FUNCTION_BLOCK FB_PowerModule
VAR_IN_OUT CONSTANT
	st_params							: ST_PowerModule_params;
	st_calibration						: ST_PowerModule_Calibration;
END_VAR


VAR_INPUT
	set									: ST_PowerModule_set; //only setteable from intern powerstack function
	r_batteryDCVoltage					: REAL;
	b_enable							: BOOL;
	e_ID								: eObject_ID;
END_VAR

VAR_OUTPUT
	{attribute 'TcAnalytics'}
	get									: ST_PowerModule_get;
	b_MccbEDM							: BOOL;
END_VAR	

VAR									
	Inverter							: FB_PowerModule_Inverter();
	Buscoupler							: FB_PowerModule_Buscoupler();
	ton_ResetPulse						: TON := (PT:= T#100MS);
	
	r_Prq: REAL;
	r_Qrq: REAL;
	pin: REAL;
	QIN: REAL;
END_VAR

IF b_enable THEN
	get.b_online := get.ui_buscouplerCommStatus = 0 AND get.ui_InverterCommStatus = 0;
	
	//Instantiate function blocks
	Buscoupler(get:=get, b_MccbEDM := b_MccbEDM, b_D7SyncRq := set.b_D7SyncRequest);
	Inverter(set := set, get:=get, st_params:=st_params);
	//defaults
	Inverter.ControlWord.b_FieldbusControlEnable := st_params.b_FieldBusControlEnable;

	//Control fan contactor.
	FanControl(st_params := st_params);
	
	//Set PowerModule status
	GetPowerModuleStatus();
	
	//Set DroopLimit
	SetInverterSettings();
	
	//Calculate derivatives
	CalculateDerivativePowerValues();
	
	//Parallel Drive
	SetParallelDrive();
	
	//setEvents
	SetEvents(events := get.Events, st_params:=st_Params);
	
	//FILL GET STRUCT
	GetInverterModes();
	FillAdditionalGets(get, set);
	
	//inverter.ControlWord.b_Reset := FALSE;
	
	SetParallelDrive();
	
	IF get.StatusWord.b_Fault THEN
		Shutdown(TRUE);
	END_IF
	
	IF GVL.b_initCycle THEN
		init();
	END_IF
END_IF

r_Prq := CompensationCurve(PIN := pin, QIN := qin, coef := st_calibration.PCoefficients, mode := 0);
r_Qrq := CompensationCurve(PIN := pin, QIN := qin, coef := st_calibration.QCoefficients, mode := 1);

METHOD BaseValueToRef : REAL;
VAR_INPUT
	IN : REAL;
END_VAR
BaseValueToRef:= IN / MAX(1, st_params.r_InverterRatedCurrent) * 100;
END_METHOD

METHOD PRIVATE CalculateDerivativePowerValues : BOOL
get.r_ReactivePower	:= get.r_ACVoltageD7 * 1.73 * get.r_ReactiveCurrent / 1000; // kvar
get.r_ActivePower	:= get.r_ACVoltageSupply* 1.73 * get.r_activeCurrent / 1000;
get.r_ApparentPower	:= SQRT(MAX(0,EXPT(get.r_ActivePower,2) + EXPT(get.r_ReactivePower,2)));
get.r_LoadPercent	:= get.r_ACCurrent / MAX(1, st_params.r_InverterRatedCurrent) * 100;
get.r_DCPower		:= get.r_DCCurrent * get.r_DCVoltage / 1000; // kW
END_METHOD

METHOD CheckDCVoltage : BOOL

VAR_INST
	b_DCprechargeOK				: BOOL; 
	b_DCVoltageOK				: BOOL;
	ton_DCOKreleaseTime			: TON := (PT:= T#1S);
END_VAR
b_DCPrechargeOK := ABS(r_BatteryDCVoltage - get.r_DCVoltage) <=  st_params.ui_DCVoltageDeltaPrechargeOK;
b_DCVoltageOK := get.r_DCVoltage > st_params.ui_DCvoltageMinPrechargeOK;

ton_DCOKReleaseTime(IN:= b_DCPrechargeOK AND b_DCVoltageOK);

CheckDCVoltage :=ton_DCOKReleaseTime.Q;
END_METHOD

METHOD CompensationCurve : REAL
VAR_INPUT
	PIN			: REAL; 
	QIN			: REAL;
	mode		: BYTE; // 0 = Pout, 1 = Qout;
END_VAR

VAR_IN_OUT CONSTANT
	coef : ST_Powermodule_PowerCurveCoefficients;
END_VAR

VAR_INST
	Q1			: REAL;
	Q2			: REAL;
	disc 		: REAL;
	Avalues		: REAL;
	Bvalues		: REAL;
	Cvalues		: REAL;
	depVar		: REAL;
	indepVar	: REAL;
END_VAR
IF NOT coef.enable THEN
	CompensationCurve := SEL(mode =0, Qin, Pin);
	RETURN; // Geen reële oplossing
END_IF


IF mode = 0 THEN
	indepVar := Pin;
	depVar := Qin;

ELSE
	indepVar := Qin;
	depVar := Pin;
END_IF

Avalues := coef.a;
BValues := coef.c*depVar + coef.d;
CValues := coef.b*EXPT(depVar,2)+coef.e*depVar + coef.f - indepVar;

disc := EXPT(BValues,2)-(4*AValues*CValues);
IF disc < 0 THEN
	CompensationCurve := indepVar;
	RETURN; // Geen reële oplossing
END_IF

// Controleer discriminant
IF Avalues = 0 THEN
    // Lineaire oplossing: B * P + C = 0 → P = -C / B
    IF BValues = 0 THEN
        RETURN; // onoplosbaar
    ELSE
        CompensationCurve := -CValues / BValues;
        RETURN;
    END_IF
END_IF

// Kwadratische oplossing (ABC)
Q1 := (-BValues + SQRT(disc)) / (2 * Avalues);
Q2 := (-BValues - SQRT(disc)) / (2 * Avalues);
CompensationCurve := Q1;
//// Kies de beste wortel (voorbeeld: dichtsbijzijnde bij indepVar)
//IF ABS(Q1 - indepVar) < ABS(Q2 - indepVar) THEN
//    CompensationCurve := Q1;
//ELSE
//    CompensationCurve := Q2;
//END_IF
END_METHOD

METHOD PRIVATE CoupleDC : BOOL
VAR_INPUT
END_VAR
IF get.StatusWord.b_ReadyToDCCharge THEN
	buscoupler.b_DCprechargeContactor := TRUE;
	buscoupler.b_DCMainContactor := CheckDCvoltage();
	CoupleDC := get.b_DCcontactorFb;
END_IF
END_METHOD

METHOD PRIVATE DecoupleDC : BOOL

VAR_INST
	b_DCmainreleaseConditionOK 	:  BOOL;
	b_DCprereleaseConditionOK 	:  BOOL;
	ton_PrechargeReleaseDelay	:  TON := (PT:= T#1S);
END_VAR

VAR
	r_DCreleaseCurrent		: REAL := 5;
	r_DCreleaseVoltage		: REAL := 10;
END_VAR
// Release main contactor first based on current
b_DCmainreleaseConditionOK := ABS(get.r_DCCurrent) < r_DCreleaseCurrent AND NOT get.StatusWord.b_Running;
IF b_DCmainreleaseConditionOK THEN
	buscoupler.b_DCmainContactor := FALSE;
END_IF

// release precharge based on voltage contactor 
b_DCprereleaseConditionOK := NOT get.b_DCcontactorFb OR r_batteryDCVoltage < r_DCreleaseVoltage; //NOT get.b_DCcontactorFb (Not for units without precharge, rewire output4 to input 4 of buscoupler.)
ton_PrechargeReleaseDelay(IN:= b_DCprereleaseConditionOK); //some delay added to be sure
IF ton_PrechargeReleaseDelay.Q THEN
	buscoupler.b_DCprechargeContactor := FALSE;
END_IF 

//Give feedback
IF b_DCprereleaseConditionOK AND b_DCmainreleaseConditionOK THEN
	DecoupleDc := NOT buscoupler.b_DCprechargeContactor AND NOT get.b_DCcontactorFb;
END_IF
END_METHOD

METHOD PRIVATE FanControl : BOOL
VAR_IN_OUT CONSTANT
	st_params : ST_Powermodule_params;
END_VAR
	


VAR_INST
	b_fanOn				: BOOL;
	tof_FanOffDelay		: TOF := (PT := T#60S);
END_VAR
IF get.r_TemperatureMax > st_params.r_TempFanOn OR get.r_LoadPercent > st_params.r_powerLoadFanOn THEN
	b_fanOn := TRUE;
ELSIF get.r_TemperatureMax < st_params.r_TempFanOn - 5 AND get.r_LoadPercent < st_params.r_powerLoadFanOn - 10 THEN
	b_fanOn := FALSE;
END_IF


tof_FanOffDelay(
	IN:= b_fanOn);
	
buscoupler.b_FanOn := set.b_FanContactor OR tof_FanOffDelay.Q;
END_METHOD

METHOD FillAdditionalGets : BOOL
VAR_IN_OUT
		get : ST_Powermodule_get;
		set	: ST_Powermodule_set;
END_VAR
get.r_TemperatureMax := GetMaxTemperature();
get.r_Pset := set.r_ActivePower;
get.r_Qset := set.r_ReactivePower;
get.b_PrechargeContactor := buscoupler.b_DCprechargeContactor;
END_METHOD

METHOD GetDiagnostics 
VAR_IN_OUT
	AddError		: ARRAY [*] OF FB_AddErrorST;
	a_ActiveEvents	: ARRAY [*] OF ST_ErrorStruct;
	w_Index			: WORD;
END_VAR

VAR
	by_errCt	: BYTE;
	by_warnCt	: BYTE;
END_VAR


VAR_INST
	b_test: BOOL;
END_VAR
(*POWERMODULE*)
	//Inverter faults
	(*OverCurr Fault*)		AddError[w_Index](
			b_ErrorTrig			:= Get.Events.b_F1OverCurrent,
			out_ST_Error			:= a_ActiveEvents[w_Index],
			w_ErrorID					:= 1,
			e_objectID				:= e_ID,
			s_Message				:= 'overcurrent fault (F1)',
			e_sev					:= eSeverity.Quickshutdown,
			);
		IF AddError[w_Index].b_out THEN by_errCt := by_errCt + 1; END_IF;
		w_Index := w_Index +1;
		
	(*OverVolt Fault*)		AddError[w_Index](
			b_ErrorTrig			:= Get.Events.b_F2OverVoltage,
			out_ST_Error			:= a_ActiveEvents[w_Index],
			w_ErrorID					:= 2,
			s_Message				:= 'DC overvoltage fault (F2)',
			e_sev					:= eSeverity.Quickshutdown,
			);
		IF AddError[w_Index].b_out THEN by_errCt := by_errCt + 1; END_IF;
		w_Index := w_Index +1;
	
	(*UnderVolt Fault*)		AddError[w_Index](
			b_ErrorTrig			:= Get.Events.b_F9UnderVoltage,
			out_ST_Error			:= a_ActiveEvents[w_Index],
			w_ErrorID					:= 3,
			s_Message				:= 'DC undervoltage fault (F9)',
			e_sev					:= eSeverity.Quickshutdown,
			);
		IF AddError[w_Index].b_out THEN by_errCt := by_errCt + 1; END_IF;
		w_Index := w_Index +1;
	
	(*ShortCurr Fault*)		AddError[w_Index](
			b_ErrorTrig		:= Get.Events.b_F91ShortCircuit,
			out_ST_Error			:= a_ActiveEvents[w_Index],
			w_ErrorID					:= 4,
			s_Message				:= 'short circuit fault (F91)',
			e_sev					:= eSeverity.Quickshutdown,
			);
		IF AddError[w_Index].b_out THEN by_errCt := by_errCt + 1; END_IF;
		w_Index := w_Index +1;
		
	(*Earth Fault*)			AddError[w_Index](
			b_ErrorTrig		:= Get.Events.b_F3EarthFault,
			out_ST_Error			:= a_ActiveEvents[w_Index],
			w_ErrorID					:= 5,
			s_Message				:= 'earth fault (F3)',
			e_sev					:= eSeverity.Quickshutdown,
			);
		IF AddError[w_Index].b_out THEN by_errCt := by_errCt + 1; END_IF;
		w_Index := w_Index +1;
		
	(*LineSync Fault*)		AddError[w_Index](
			b_ErrorTrig		:= Get.Events.b_F10LineSynchFault,
			out_ST_Error			:= a_ActiveEvents[w_Index],
			w_ErrorID					:= 6,
			s_Message				:= 'line synchronisation fault (F10)',
			e_sev					:= eSeverity.Quickshutdown,
			);
		IF AddError[w_Index].b_out THEN by_errCt := by_errCt + 1; END_IF;
		w_Index := w_Index +1;
	
	(*Keypad Fault*)		AddError[w_Index](
			b_ErrorTrig		:= Get.Events.b_F52KeypadOCCommFault,
			out_ST_Error			:= a_ActiveEvents[w_Index],
			w_ErrorID					:= 7,
			s_Message				:= 'keypad communication fault (F52)',
			e_sev					:= eSeverity.warning,
			);
		IF AddError[w_Index].b_out THEN by_errCt := by_errCt + 1; END_IF;
		w_Index := w_Index +1;
	
	(*Fieldbus Fault*)		AddError[w_Index](
			b_ErrorTrig		:= Get.Events.b_F53FieldbusFault,
			out_ST_Error			:= a_ActiveEvents[w_Index],
			w_ErrorID					:= 8,
			s_Message				:= 'fieldbus fault (F53)',
			e_sev					:= eSeverity.Quickshutdown,
			);
		IF AddError[w_Index].b_out THEN by_errCt := by_errCt + 1; END_IF;
		w_Index := w_Index +1;
		
	(*Systembus Fault*)		AddError[w_Index](
			b_ErrorTrig		:= Get.Events.b_F59SystembusFault,
			out_ST_Error			:= a_ActiveEvents[w_Index],
			w_ErrorID					:= 9,
			s_Message				:= 'system bus Fault (F59)',
			e_sev					:= eSeverity.Quickshutdown,
			);
		IF AddError[w_Index].b_out THEN by_errCt := by_errCt + 1; END_IF;
		w_Index := w_Index +1;
	
	(*IOslot Fault*)		AddError[w_Index](
			b_ErrorTrig		:= Get.Events.b_F54SlotCommunicationFault,
			out_ST_Error			:= a_ActiveEvents[w_Index],
			w_ErrorID					:= 10,
			s_Message				:= 'IO slot communication fault (F54)',
			e_sev					:= eSeverity.Quickshutdown,
			);
		IF AddError[w_Index].b_out THEN by_errCt := by_errCt + 1; END_IF;
		w_Index := w_Index +1;
		
	(*4ma meas Fault*)		AddError[w_Index](
			b_ErrorTrig		:= Get.Events.b_F50Meas4mAFault,
			out_ST_Error			:= a_ActiveEvents[w_Index],
			w_ErrorID					:= 11,
			s_Message				:= 'measurement 4 mA fault (F50)',
			e_sev					:= eSeverity.info,
			b_AutoClear			:= TRUE,
		);
		w_Index := w_Index +1;
		
	(*Watchdog Fault*)		AddError[w_Index](
			b_ErrorTrig		:= Get.Events.b_WatchdogError,
			out_ST_Error			:= a_ActiveEvents[w_Index],
			w_ErrorID					:= 12,
			s_Message				:= 'watchdog fault',
			e_sev					:= eSeverity.Quickshutdown,
			);
		IF AddError[w_Index].b_out THEN by_errCt := by_errCt + 1; END_IF;
		w_Index := w_Index +1;
	
	(*Mccb Trip*)			AddError[w_Index](
			b_ErrorTrig			:= FALSE, //Get.Events.b_MCCBtrip,
			out_ST_Error			:= a_ActiveEvents[w_Index],
			w_ErrorID					:= 13,
			s_Message				:= 'MCCB trip',
			e_sev					:= eSeverity.warning
		);
		w_Index := w_Index +1;

	(*Shutdown TimeOut*)			AddError[w_Index](
			b_ErrorTrig			:= Get.Events.b_ShutdownTimeOut,
			out_ST_Error			:= a_ActiveEvents[w_Index],
			w_ErrorID					:= 14,
			s_Message				:= 'shutdown Timeout',
			e_sev					:= eSeverity.QuickShutdown
		);
		w_Index := w_Index +1;
		
	(*output phase fault (F11)*)	AddError[w_Index](
			b_ErrorTrig				:= Get.Events.b_F11OutputPhaseFault,
			out_ST_Error			:= a_ActiveEvents[w_Index],
			w_ErrorID				:= 15,
			s_Message				:= 'output phase fault (F11)',
			e_sev					:= eSeverity.Quickshutdown
		);
		w_Index := w_Index +1;
		
	(*charge fault (F80)*)			AddError[w_Index](
			b_ErrorTrig				:= Get.Events.b_F80ChargeFault,
			out_ST_Error			:= a_ActiveEvents[w_Index],
			w_ErrorID				:= 16,
			s_Message				:= 'charge fault (F80)',
			e_sev					:= eSeverity.Quickshutdown
		);
		w_Index := w_Index +1;
		
		(*charge fault (F80)*)			AddError[w_Index](
			b_ErrorTrig				:= Get.Events.b_F51ExternalFault,
			out_ST_Error			:= a_ActiveEvents[w_Index],
			w_ErrorID				:= 17,
			s_Message				:= 'external fault (F51)',
			e_sev					:= eSeverity.Quickshutdown
		);
		w_Index := w_Index +1;
		
		(*IGBT fault (F31)*)		AddError[w_Index](
			b_ErrorTrig				:= Get.Events.b_F31IGBTFault,
			out_ST_Error			:= a_ActiveEvents[w_Index],
			w_ErrorID				:= 18,
			s_Message				:= 'IGBT fault (F31)',
			e_sev					:= eSeverity.Quickshutdown
		);
		w_Index := w_Index +1;
		
		(*MCB state fault (F64)*)		AddError[w_Index](
			b_ErrorTrig				:= Get.Events.b_F64MCBstateFault,
			out_ST_Error			:= a_ActiveEvents[w_Index],
			w_ErrorID				:= 19,
			s_Message				:= 'MCB state fault (F64)',
			e_sev					:= eSeverity.Quickshutdown
		);
		w_Index := w_Index +1;
	
	//Temperature Faults
	(*Gridch L1 Alarm*)		AddError[w_Index](
			b_ErrorTrig		:= Get.Events.b_CMChokeTemperatureTooHigh[1],
			out_ST_Error			:= a_ActiveEvents[w_Index],
			w_ErrorID					:= 20 ,
			s_Message				:= 'gridchoke L1 temperature too high',
			e_sev					:= eSeverity.normalshutdown,
			);
		IF AddError[w_Index].b_out THEN by_errCt := by_errCt + 1; END_IF;
		w_Index := w_Index +1;
		
	(*Gridch L2 Alarm*)		AddError[w_Index](
			b_ErrorTrig		:= Get.Events.b_CMChokeTemperatureTooHigh[2], //phase 2
			out_ST_Error			:= a_ActiveEvents[w_Index],
			w_ErrorID					:= 21 ,
			s_Message				:= 'gridchoke L2 temperature too high',
			e_sev					:= eSeverity.normalshutdown,
			);
		IF AddError[w_Index].b_out THEN by_errCt := by_errCt + 1; END_IF;
		w_Index := w_Index +1;
		
	(*Gridch L3 Alarm*)		AddError[w_Index](
			b_ErrorTrig		:= Get.Events.b_CMChokeTemperatureTooHigh[3], //phase 3
			out_ST_Error			:= a_ActiveEvents[w_Index],
			w_ErrorID					:= 22 ,
			s_Message				:= 'gridchoke L3 temperature too high',
			e_sev					:= eSeverity.normalshutdown,
			);
		IF AddError[w_Index].b_out THEN by_errCt := by_errCt + 1; END_IF;
		w_Index := w_Index +1;
		
	(*CMch L1 Alarm*)		AddError[w_Index](
			b_ErrorTrig		:= Get.Events.b_GridChokeTemperatureTooHigh[1], //phase 1
			out_ST_Error			:= a_ActiveEvents[w_Index],
			w_ErrorID					:= 23 ,
			s_Message				:= 'CM choke L1 temperature too high',
			e_sev					:= eSeverity.normalshutdown,
			);
		IF AddError[w_Index].b_out THEN by_errCt := by_errCt + 1; END_IF;
		w_Index := w_Index +1;
		
	(*CMch L2 Alarm*)		AddError[w_Index](
			b_ErrorTrig		:= Get.Events.b_CMChokeTemperatureTooHigh[2], //phase 2
			out_ST_Error			:= a_ActiveEvents[w_Index],
			w_ErrorID					:= 24 ,
			s_Message				:= 'CM choke L2 temperature too high',
			e_sev					:= eSeverity.normalshutdown,
			);
		IF AddError[w_Index].b_out THEN by_errCt := by_errCt + 1; END_IF;
		w_Index := w_Index +1;
		
	(*CMch L3 Alarm*)		AddError[w_Index](
			b_ErrorTrig		:= Get.Events.b_CMChokeTemperatureTooHigh[3], //phase 3
			out_ST_Error			:= a_ActiveEvents[w_Index],
			w_ErrorID					:= 25 ,
			s_Message				:= 'CM choke L3 temperature too high',
			e_sev					:= eSeverity.normalshutdown,
			);
		IF AddError[w_Index].b_out THEN by_errCt := by_errCt + 1; END_IF;
		w_Index := w_Index +1;
		
	(*CMch DC Alarm*)		AddError[w_Index](
			b_ErrorTrig		:= Get.Events.b_CMChokeTemperatureTooHigh[4], //DC
			out_ST_Error			:= a_ActiveEvents[w_Index],
			w_ErrorID					:= 26 ,
			s_Message				:= 'CM choke DC temperature too high',
			e_sev					:= eSeverity.normalshutdown,
			);
		IF AddError[w_Index].b_out THEN by_errCt := by_errCt + 1; END_IF;
		w_Index := w_Index +1;
		
	(*Inverter Alarm*)		AddError[w_Index](
			b_ErrorTrig		:= Get.Events.b_F14UnitOverTemperature,
			out_ST_Error			:= a_ActiveEvents[w_Index],
			w_ErrorID					:= 27 ,
			s_Message				:= 'overtemperature fault (F14)',
			e_sev					:= eSeverity.Quickshutdown
		);
		IF AddError[w_Index].b_out THEN by_errCt := by_errCt + 1; END_IF;
		w_Index := w_Index +1;	
		
	(*PT100 Fault*)			AddError[w_Index](
			b_ErrorTrig		:= Get.Events.b_F56TemperatureFault, //inverter Pt100 measurement
			out_ST_Error			:= a_ActiveEvents[w_Index],
			w_ErrorID					:= 28 ,
			s_Message				:= 'pt100 temperature fault (F56)',
			e_sev					:= eSeverity.normalshutdown,
			);
		IF AddError[w_Index].b_out THEN by_errCt := by_errCt + 1; END_IF;
		w_Index := w_Index +1;
		
	
	//Temperature Warnings
	(*Gridch L1 Warning*)	AddError[w_Index](
			b_ErrorTrig			:= Get.Events.b_gridChokeTemperatureHigh[1], //phase 1
			out_ST_Error			:= a_ActiveEvents[w_Index],
			w_ErrorID					:= 40 ,
			s_Message				:= 'gridchoke L1 temperature high',
			e_sev					:= eSeverity.warning,
			b_AutoClear			:= TRUE,
			);
		IF AddError[w_Index].b_out THEN by_warnCt := by_warnCt + 1; END_IF;
		w_Index := w_Index +1;
		
	(*Gridch L2 Warning*)	AddError[w_Index](
			b_ErrorTrig		:= Get.Events.b_GridchokeTemperatureHigh[2], //phase 2
			out_ST_Error			:= a_ActiveEvents[w_Index],
			w_ErrorID					:= 41 ,
			s_Message				:= 'gridchoke L2 temperature high',
			e_sev					:= eSeverity.warning,
			b_AutoClear			:= TRUE,
			);
		IF AddError[w_Index].b_out THEN by_warnCt := by_warnCt + 1; END_IF;
		w_Index := w_Index +1;
		
	(*Gridch L3 Warning*)	AddError[w_Index](
			b_ErrorTrig		:= Get.Events.b_GridChokeTemperatureHigh[3], //phase 3
			out_ST_Error			:= a_ActiveEvents[w_Index],
			w_ErrorID					:= 42 ,
			s_Message				:= 'gridchoke L3 temperature high',
			e_sev					:= eSeverity.warning,
			b_AutoClear			:= TRUE,
			);
		IF AddError[w_Index].b_out THEN by_warnCt := by_warnCt + 1; END_IF;
		w_Index := w_Index +1;
		
	(*CMch L1 Warning*)		AddError[w_Index](
			b_ErrorTrig		:= Get.Events.b_CMChokeTemperatureHigh[1], //phase 1
			out_ST_Error			:= a_ActiveEvents[w_Index],
			w_ErrorID					:= 43 ,
			s_Message				:= 'CM choke L1 temperature high',
			e_sev					:= eSeverity.warning,
			b_AutoClear			:= TRUE,
			);
		IF AddError[w_Index].b_out THEN by_warnCt := by_warnCt + 1; END_IF;
		w_Index := w_Index +1;
		
	(*CMch L2 Warning*)		AddError[w_Index](
			b_ErrorTrig		:= Get.Events.b_CMChokeTemperatureHigh[2], //phase 2
			out_ST_Error			:= a_ActiveEvents[w_Index],
			w_ErrorID				:= 44 ,
			s_Message				:= 'CM choke L2 temperature high',
			e_sev					:= eSeverity.warning,
			b_AutoClear			:= TRUE,
			);
		IF AddError[w_Index].b_out THEN by_warnCt := by_warnCt + 1; END_IF;
		w_Index := w_Index +1;
		
	(*CMch L3 Warning*)		AddError[w_Index](
			b_ErrorTrig		:= Get.Events.b_CMChokeTemperatureHigh[3], //phase 3
			out_ST_Error			:= a_ActiveEvents[w_Index],
			w_ErrorID					:= 45 ,
			s_Message				:= 'CM choke L3 temperature high',
			e_sev					:= eSeverity.warning,
			b_AutoClear			:= TRUE,
			);
		IF AddError[w_Index].b_out THEN by_warnCt := by_warnCt + 1; END_IF;
		w_Index := w_Index +1;
		
	(*CMch DC Warning*)		AddError[w_Index](
			b_ErrorTrig		:= Get.Events.b_CMChokeTemperatureHigh[4], //DC
			out_ST_Error			:= a_ActiveEvents[w_Index],
			w_ErrorID					:= 46 ,
			s_Message				:= 'CM choke DC temperature high',
			e_sev					:= eSeverity.warning,
			b_AutoClear			:= TRUE,
			);
		IF AddError[w_Index].b_out THEN by_warnCt := by_warnCt + 1; END_IF;
		w_Index := w_Index +1;
		
	(*Inverter Warning*)	AddError[w_Index](
			b_ErrorTrig			:= Get.Events.b_inverterTemperatureHigh, //inverter
			out_ST_Error			:= a_ActiveEvents[w_Index],
			w_ErrorID					:= 47 ,
			s_Message				:= 'Inverter temperature high',
			e_sev					:= eSeverity.warning,
			b_AutoClear			:= TRUE,
			);
		IF AddError[w_Index].b_out THEN by_warnCt := by_warnCt + 1; END_IF;
		w_Index := w_Index +1;
		
	(*PT100 Range Warning*)	AddError[w_Index](
			b_ErrorTrig			:= Get.Events.b_CMSTemperatureRangeWarning, //inverter Pt100 measurement
			out_ST_Error			:= a_ActiveEvents[w_Index],
			w_ErrorID					:= 48 ,
			s_Message				:= 'CMS pt100 temperature range warning',
			e_sev					:= eSeverity.warning,
			b_AutoClear			:= TRUE,
			);
		IF AddError[w_Index].b_out THEN by_warnCt := by_warnCt + 1; END_IF;
		w_Index := w_Index +1;
		
	(*FanState Warning*)	AddError[w_Index](
			b_ErrorTrig			:= Get.Events.b_FanStateUnknownWarning, //general warning from inverter
			out_ST_Error			:= a_ActiveEvents[w_Index],
			w_ErrorID					:= 61 ,
			s_Message				:= 'fan state warning',
			e_sev					:= eSeverity.warning,
			t_triggerTime			:= T#1S,
			b_AutoClear				:= TRUE,
			);
		IF AddError[w_Index].b_out THEN by_warnCt := by_warnCt + 1; END_IF;
		w_Index := w_Index +1;
	
	(*PT100Underrange*)	AddError[w_Index](
			b_ErrorTrig			:= Get.Events.b_PT100Underrange, //general warning from inverter
			out_ST_Error			:= a_ActiveEvents[w_Index],
			w_ErrorID					:= 62 ,
			s_Message				:= 'PT100 underrange warning',
			e_sev					:= eSeverity.warning,
			b_AutoClear			:= TRUE,
			);
		IF AddError[w_Index].b_out THEN by_warnCt := by_warnCt + 1; END_IF;
		w_Index := w_Index +1;
		
	(*PT100Overrange*)	AddError[w_Index](
			b_ErrorTrig			:= Get.Events.b_PT100Underrange, //general warning from inverter
			out_ST_Error			:= a_ActiveEvents[w_Index],
			w_ErrorID					:= 63 ,
			s_Message				:= 'PT100 Overrange warning',
			e_sev					:= eSeverity.warning,
			b_AutoClear			:= TRUE,
			);
		IF AddError[w_Index].b_out THEN by_warnCt := by_warnCt + 1; END_IF;
		w_Index := w_Index +1;

	(*PT100 Error*)	AddError[w_Index](
			b_ErrorTrig			:= Get.Events.by_PT100ErrorCount > 5, //general warning from inverter
			out_ST_Error			:= a_ActiveEvents[w_Index],
			w_ErrorID					:= 64 ,
			s_Message				:= 'more than 5 PT100 errors',
			e_sev					:= eSeverity.Normalshutdown,
			b_AutoClear			:= TRUE,
			);
		IF AddError[w_Index].b_out THEN by_errCt := by_errCt + 1; END_IF;
		w_Index := w_Index +1;
		
	(*Buscoupler comm error*)	AddError[w_Index](
			b_ErrorTrig			:= Get.ui_BuscouplerCommStatus <>0, //general warning from inverter
			out_ST_Error			:= a_ActiveEvents[w_Index],
			w_ErrorID					:= 65 ,
			s_Message				:= 'buscoupler communication error',
			e_sev					:= eSeverity.Normalshutdown,
			);
		IF AddError[w_Index].b_out THEN by_errCt := by_errCt + 1; END_IF;
		w_Index := w_Index +1;
	
	(*Inverter comm error*)	AddError[w_Index](
			b_ErrorTrig			:= Get.ui_InverterCommStatus <>0 AND Get.ui_InverterCommStatus <15, //general warning from inverter
			out_ST_Error			:= a_ActiveEvents[w_Index],
			w_ErrorID					:= 66 ,
			s_Message				:= 'inverter communication error',
			e_sev					:= eSeverity.Quickshutdown
			);
		IF AddError[w_Index].b_out THEN by_errCt := by_errCt + 1; END_IF;
		w_Index := w_Index +1;
		
	(*Inverter temp throttling active*)	AddError[w_Index](
			b_ErrorTrig			:= get.Events.b_TempThrottlingActive, //general warning from inverter
			out_ST_Error			:= a_ActiveEvents[w_Index],
			w_ErrorID					:= 67 ,
			s_Message				:= 'temperature throttling active',
			e_sev					:= eSeverity.Warning,
			b_AutoClear			:= TRUE,
			);
		IF AddError[w_Index].b_out THEN by_warnCt := by_warnCt + 1; END_IF;
		w_Index := w_Index +1;
		
	(*Inverter current throttling active*)	AddError[w_Index](
			b_ErrorTrig			:= get.Events.b_CurrThrottlingActive, //general warning from inverter
			out_ST_Error			:= a_ActiveEvents[w_Index],
			w_ErrorID					:= 68 ,
			s_Message				:= 'Current throttling active',
			e_sev					:= eSeverity.Warning,
			b_AutoClear			:= TRUE,
			);
		IF AddError[w_Index].b_out THEN by_warnCt := by_warnCt + 1; END_IF;
		w_Index := w_Index +1;
		
		(*Inverter current throttling active*)	AddError[w_Index](
			b_ErrorTrig			:= get.StatusWord.b_Fault, //general warning from inverter
			out_ST_Error			:= a_ActiveEvents[w_Index],
			w_ErrorID					:= 69,
			s_Message				:= 'General fault',
			e_sev					:= eSeverity.Quickshutdown,
			);
		IF AddError[w_Index].b_out THEN by_errCt := by_errCt + 1; END_IF;
		w_Index := w_Index +1;
		
		(*UVR fault*)			AddError[w_Index](
			b_ErrorTrig				:= Get.Events.b_24VdcUVRFault,
			out_ST_Error			:= a_ActiveEvents[w_Index],
			w_ErrorID				:= 70,
			s_Message				:= 'UVR 24VDC Fault',
			e_sev					:= eSeverity.warning,
			b_AutoClear				:= TRUE,
		);
		w_Index := w_Index +1;

			

get.events.b_GeneralFaultFlag := by_errCt <> 0;
get.events.b_GeneralWarningFlag := by_warnCt <>0;
END_METHOD

METHOD PRIVATE GetInverterModes
IF get.UgridStatusWord.b_AFEmodeActive THEN
	get.e_InverterMode := eInvertermodes.afe;
ELSIF get.UgridStatusWord.b_IslandModeActive OR get.UgridStatusWord.b_MicrogridModeActive AND get.r_FrequencyDroop <= 0.1 THEN
	get.e_InverterMode := eInvertermodes.Island;	
ELSE
	get.e_InverterMode := eInvertermodes.Microgrid;
END_IF
END_METHOD

METHOD PRIVATE GetMaxTemperature : REAL;
// calculate max
GetMaxTemperature := MAX(
						get.r_TemperatureCMChoke[1], 
						get.r_TemperatureCMChoke[2], 
						get.r_TemperatureCMChoke[3], 
						get.r_TemperatureCMChoke[4],
						get.r_TemperatureGridChoke[1], 
						get.r_TemperatureGridChoke[2], 
						get.r_TemperatureGridChoke[3]
);
END_METHOD

METHOD PRIVATE GetPowerModuleStatus : BOOL
IF get.StatusWord.b_Fault OR get.Events.b_GeneralFaultFlag THEN
	get.e_Status := eStatusPowerModule.fault;
ELSIF get.StatusWord.b_Running THEN
	get.e_Status := eStatusPowermodule.running;
ELSIF get.StatusWord.b_ReadyToOperate THEN
	get.e_Status := eStatusPowermodule.idle;
ELSIF get.StatusWord.b_DCAtReference THEN	
	get.e_Status := eStatusPowermodule.DcOK;
ELSIF get.StatusWord.b_ReadyToDCCharge THEN
	get.e_Status := eStatusPowermodule.off;
ELSE
	get.e_Status := eStatusPowermodule.Init;
END_IF
END_METHOD

METHOD GetTemperatureEvents : BOOL
VAR_INPUT
	Warnings	: 	BOOL;
END_VAR
IF Warnings THEN
	GetTemperatureEvents := get.Events.b_CMChokeTemperatureHigh[1] 	OR
			get.Events.b_CMChokeTemperatureHigh[2]		OR
			get.Events.b_CMChokeTemperatureHigh[3]		OR
			get.Events.b_CMChokeTemperatureHigh[4] 		OR
			get.Events.b_GridChokeTemperatureHigh[1]	OR
			get.Events.b_GridChokeTemperatureHigh[2]	OR
			get.Events.b_GridChokeTemperatureHigh[3]	OR
			get.Events.b_inverterTemperatureHigh;
ELSE
	GetTemperatureEvents := get.Events.b_CMChokeTemperatureTooHigh[1] 	OR
			get.Events.b_CMChokeTemperatureTooHigh[2]	OR
			get.Events.b_CMChokeTemperatureTooHigh[3]	OR
			get.Events.b_CMChokeTemperatureTooHigh[4]	OR
			get.Events.b_GridChokeTemperatureTooHigh[1]	OR
			get.Events.b_GridChokeTemperatureTooHigh[2]	OR
			get.Events.b_GridChokeTemperatureTooHigh[3]	OR
			get.Events.b_F56TemperatureFault;
END_IF
END_METHOD

METHOD Idle : BOOL
//Inverter.controlWord.b_ChargeDC := TRUE;
//inverter.ControlWord.b_run := TRUE;

//Set powermode
inverter.powermode := ePowermodes.Droop;
inverter.r_BaseCurrentRef := 0;
inverter.r_ReactiveCurrentRef := 0;
SetVoltageFrequency(SetToIn := TRUE, VoltIN := settings.GridParams.r_GridNominalVoltage, FreqIn := settings.GridParams.r_GridNominalFrequency);
inverter.startMode := FALSE;
inverter.Island(TRUE);
Idle := get.StatusWord.b_readytooperate AND NOT get.GridcodeStatusWord.b_GridCodeTripActive;
END_METHOD

METHOD init : BOOL

VAR_INST
	
END_VAR
inverter.ControlWord.b_ChargeDC := FALSE;
inverter.ControlWord.b_run := FALSE;
inverter.ControlWord.b_Reset := TRUE;
END_METHOD

METHOD Reset : BOOL
ton_ResetPulse(IN:= NOT ton_ResetPulse.Q);
set.b_QuickstopInactive := TRUE;

Inverter.ControlWord.b_Reset := TRUE;
buscoupler.b_MCCBChargeSpring := TRUE;

IF NOT (get.events.b_GeneralFaultFlag OR get.StatusWord.b_Fault) THEN
	Inverter.ControlWord.b_Reset := FALSE;
	buscoupler.b_MCCBChargeSpring := FALSE;
END_IF

Reset := get.e_Status <> eStatusPowerModule.fault;
END_METHOD

METHOD Run : BOOL
VAR_INPUT
	Powermode			: ePowermodes;
	InverterMode		: EInvertermodes;
	InternalPowerSet		: BOOL;
END_VAR

VAR_INST
	r_DroopMin			: REAL;
	r_DroopMax			: REAL;
END_VAR
//Set powermodes
inverter.Powermode := powermode;
inverter.startMode := FALSE;


// set invertermode
CASE InverterMode OF
	eInverterModes.Afe : Inverter.AFE();
	eInverterModes.Microgrid : Inverter.Microgrid();
	eInverterModes.Island : Inverter.Island(FALSE);
END_CASE

SetVoltageFrequency(InternalPowerSet, set.r_NomVoltage, set.r_NomFrequency);

//Set absolute power and current limits of inverter
IF InternalPowerSet THEN
	inverter.r_InputActiveCurrentLimit := 100;
	inverter.r_OutputActiveCurrentLimit := 100;
	Inverter.Island(TRUE);
ELSE
	SetInverterRefs_Limits(get := get, set := set, 
		r_InputActiveCurrentLimitRef => inverter.r_InputActiveCurrentLimit,
		r_OutputActiveCurrentLimitRef => inverter.r_OutputActiveCurrentLimit,
		r_basecurrentref => inverter.r_BaseCurrentRef,
		r_ReactiveCurrentRef => inverter.r_ReactiveCurrentRef
	);
END_IF

inverter.ControlWord.b_run := TRUE;
run := get.StatusWord.b_Running;
END_METHOD

METHOD PRIVATE SetEvents
VAR_IN_OUT CONSTANT
	st_params					: ST_Powermodule_Params;
END_VAR


VAR_IN_OUT
	events						: ST_Powermodule_events;
END_VAR

VAR 
	w_Index										: WORD;
END_VAR
FOR w_Index:=1 TO 4 DO
	 LimitTrigger(
		r_IN := get.r_TemperatureCMChoke[w_Index],
		b_HighEnable:= TRUE,
		r_HighLimit:= st_Params.r_FilterTempAlarm,
		r_HighWarning:= st_params.r_FilterTempWarning,
		b_LowEnable:= FALSE,
		r_LowLimit:= 0,
		r_LowWarning:= 0,
		r_hysteresis:= 5,
		b_Warning=> get.Events.b_CMChokeTemperatureHigh[w_Index],
		b_Fault=> get.Events.b_CMChokeTemperatureTooHigh[w_Index]
		);
END_FOR

FOR w_Index:=1 TO 3 DO
	LimitTrigger(
		r_IN := get.r_TemperatureCMChoke[w_Index],
		b_HighEnable:= TRUE,
		r_HighLimit:= st_params.r_FilterTempAlarm,
		r_HighWarning:= st_params.r_FilterTempWarning,
		b_LowEnable:= FALSE,
		r_LowLimit:= 0,
		r_LowWarning:= 0,
		r_hysteresis:= 5,
		b_Warning=>get.Events.b_GridChokeTemperatureHigh[w_Index],
		b_Fault=> get.Events.b_GridChokeTemperatureTooHigh[w_Index]
	);
END_FOR

// set warning when CMS PT100 gives out of range values. 
get.Events.b_CMSTemperatureRangeWarning := NOT get.w_TemperatureFaultWord =0;

//Set fan state warning
get.Events.b_FanStateUnknownWarning := get.b_FanFb AND NOT buscoupler.b_FanOn;
get.Events.b_24VdcUVRFault := NOT get.b_MccbUvr24VdcOK AND get.b_DCcontactorFb;
END_METHOD

METHOD PRIVATE SetInverterRefs_Limits : BOOL

VAR_IN_OUT
	get 			: ST_Powermodule_get;
	set				: ST_Powermodule_set;
END_VAR

VAR_OUTPUT
	r_InputActiveCurrentLimitRef : REAL;
	r_OutputActiveCurrentLimitRef : REAL;
	r_BaseCurrentRef			: REAL;
	r_ReactiveCurrentRef		: REAL;
END_VAR

VAR_INST
	r_PLimitOverhead				: REAL := 1.1;
	fb_ActiveCurrentMeasMA			: FB_movingAverage := (length := 1000, enable := TRUE);	
	r_MaxOvercurrentFactor			: REAL;	
	r_ActivePowerRQ					: REAL;
	r_ReactivePowerRQ				: REAL;
	fb_DynamicreactiveRemainMA		: FB_movingAverage := (length := 10, enable := TRUE);
	r_reactiveMaxCurrent			: REAL;
	r_ReactiveLimitCorrection		: REAL := 1.20;
	r_NomVoltage					: REAL := 400;
	ar_Throttling					: ARRAY [1..20] OF REAL;
	fb_SmoothThrottling				: FB_CTRL_Moving_Average := (eMode := e_ctrl_mode.eCTRL_MODE_ACTIVE);
	st_params_SmoothThrottling		: ST_CTRL_MOVING_AVERAGE_PARAMS := (
		 								tCtrlCycleTime := T#1S,
										tTaskCycleTime := T#1MS,
										nSamplesToFilter := 10);
										
	 r_InputActiveCurrentLimit		: REAL;
	 r_outputActiveCurrentLimit		: REAL;
	 r_baseCurrentSetpoint			: REAL;
	 r_reactiveCurrentsetpoint		: REAL;
	 r_VoltAC						: REAL;
	 r_DynamicCurrentLimit			: REAL;
	 r_ThrottlingValueFilterTemp	: REAL;
	 r_ThrottlingValueInverterTemp	: REAL;
	 r_ThrottlingValueMindex		: REAL;
	 r_ThrottlingActual				: REAL;
	 
	 
	 ePIDctrl						: E_CTRL_Mode;
	 //Mindex limiter
	r_ActReactiveToThrottlingValue	: REAL;
	fb_PIDMindex					: FB_CTRL_PID_EXT := (emode := e_Ctrl_mode.eCTRL_MODE_ACTIVE);
	st_Params_PIDMindex				: ST_CTRL_PID_EXT_PARAMS := ( 
										tTaskCycleTime := T#1MS,
										tCtrlCycleTime := T#1MS,
										fKp	:= 0.05,
										tTn := T#500MS,
										tTd := T#0S,
										tTv := T#0MS,
										fOutMaxLimit := 0,
										fOutMinLimit := -1,
										fouterwindow := 0
										);


	//AC current limiter
	fb_RampCurrentLimit				: FB_RAMP_Dual := (Enable := TRUE, rampDown := 50, rampUp := 20);									
	fb_PIDCurrentLimit				: FB_CTRL_PID_EXT;
	st_Params_PIDCurrentLimit		: ST_CTRL_PID_EXT_PARAMS := ( 
										tTaskCycleTime := T#1MS,
										tCtrlCycleTime := T#1MS,
										fKp	:= 0.5,
										tTn := T#500MS,
										tTd := T#0MS,
										tTv := T#0MS,
										fDeadbandInput := 10
										);
										
END_VAR
IF ton_ResetPulse.Q AND NOT get.StatusWord.b_Running THEN
	ePIDctrl := e_Ctrl_mode.eCTRL_MODE_RESET;
ELSE
	ePIDctrl := e_Ctrl_mode.eCTRL_MODE_Active;	
END_IF

r_VoltAC := get.r_ACVoltageSupply;
fb_ActiveCurrentMeasMA(IN := get.r_ActiveCurrent);
r_MaxOvercurrentFactor := MIN(st_params.r_ACCurrentLimitMax / MAX(1, st_params.r_InverterRatedCurrent), set.r_overcurrentFactor);

st_params_SmoothThrottling.pWorkArray_ADR := ADR(ar_Throttling);
st_params_SmoothThrottling.nWorkArray_SIZEOF := SIZEOF(ar_Throttling);

fb_SmoothThrottling(
	fin := get.r_TemperatureMax,
	stParams := st_params_SmoothThrottling);

r_ThrottlingValueFilterTemp := scale(
		r_in:=fb_SmoothThrottling.fOut,
		 In_min:= st_params.r_FilterTempWarning,
		 In_max:= st_params.r_FilterTempAlarm,
		 Out_min:= r_MaxOvercurrentFactor,
		 Out_max:= st_params.r_ThrottlingMinimum);
		
r_ThrottlingValueInverterTemp := scale(
		r_in:=get.r_TemperatureInverter,
		 In_min:= st_params.r_InverterTempWarning,
		 In_max:= st_params.r_InverterTempAlarm,
		 Out_min:= r_MaxOvercurrentFactor,
		 Out_max:= st_params.r_ThrottlingMinimum);	

r_ThrottlingActual	:= MIN(r_ThrottlingValueInverterTemp,r_ThrottlingValueFilterTemp);	

//TOTAL AC CURRENT LIMIT
	st_Params_PIDCurrentLimit.fOutMaxLimit := st_params.r_ACCurrentLimitMax;
	st_Params_PIDCurrentLimit.fOutMinLimit := st_params.r_ACCurrentLimitMin;
	fb_RampCurrentLimit(SetToIn := NOT get.StatusWord.b_Running, IN :=  LIMIT(st_params.r_ACcurrentLimitMin, set.r_ACcurrentLimit, st_params.r_InverterRatedCurrent *  r_throttlingActual));
	fb_PIDCurrentLimit(
		eMode := ePIDctrl,
		fSetpointValue := LIMIT(fb_RampCurrentLimit.Q,get.r_ACCurrent, fb_RampCurrentLimit.Q),
		fActualValue := get.r_ACCurrent,
		stParams:= st_params_PIDCurrentLimit,
		fout => r_DynamicCurrentLimit
		);
	
	IF fb_PIDCurrentLimit.bError THEN
		r_DynamicCurrentLimit := LIMIT(st_params.r_ACcurrentLimitMin, set.r_ACcurrentLimit, st_params.r_InverterRatedCurrent *  r_throttlingActual);
	END_IF
	
	IF st_calibration.b_StartCalibration THEN
		r_DynamicCurrentLimit := 650;
	END_IF

//ACTIVE CURRENT LIMIT
	r_InputActiveCurrentLimit := LIMIT(0 , kWToCurrent(ABS(set.r_Pmin), 400), st_params.r_ACCurrentLimitMax);
	r_OutputActiveCurrentLimit := LIMIT(0 , kWToCurrent(ABS(set.r_Pmax),  400), st_params.r_ACCurrentLimitMax);

//ACTIVE SETPOINT
	r_activePowerRQ := CompensationCurve(PIN := set.r_ActivePower, QIN := get.r_ReactivePower, coef := st_calibration.PCoefficients, mode := 0);
	r_ActivePowerRQ	:= LIMIT(get.r_Pmin, r_ActivePowerRQ, get.r_Pmax);


//REACTIVE SETPOINT + MINDEX LIMIT
st_params_PIDMindex.fDeadBandInput := st_params.r_ModulationIndexLimitHyst;
	fb_PIDMindex(
		eMode := ePIDctrl,
		fsetpointvalue :=  st_params.r_ModulationIndexLimit,
		fActualValue := get.r_ModulationIndex,
		stparams := st_Params_PIDMindex
	);	
	r_ThrottlingValueMindex := fb_PIDMindex.fout + 1;
	fb_DynamicreactiveRemainMA(IN := SQRT(MAX(EXPT(r_DynamicCurrentLimit,2) - EXPT(fb_ActiveCurrentMeasMA.Q*r_ReactiveLimitCorrection ,2), 0)) * r_ThrottlingValueMindex);
	r_ReactivePowerRQ := CompensationCurve(PIN := get.r_activePower, QIN := set.r_ReactivePower, coef := st_calibration.QCoefficients, mode := 1);
	
	//to jump to PID value when throttling starts. Otherwise takes quite some time to get there.
	r_ActReactiveToThrottlingValue := kWToCurrent(r_ActivePowerRQ, get.r_ACVoltageD7) / MAX(1, fb_DynamicreactiveRemainMA.Q);
	IF get.r_ModulationIndex > MIN(100, st_params.r_ModulationIndexLimit + st_params.r_ModulationIndexLimitHyst) AND r_ThrottlingValueMindex > r_ActReactiveToThrottlingValue THEN
		fb_PIDMindex.fManSyncValue := r_ActReactiveToThrottlingValue - 1;
		fb_PIDMindex.bSync := TRUE;
	ELSE
		fb_PIDMindex.bSync := FALSE;
	END_IF
	
//power overwrites before it is converted to refs
	IF st_calibration.b_StartCalibration THEN
		r_activePowerRQ := st_calibration.r_Pset;
		r_ReactivePowerRQ	:= st_calibration.r_Qset;
	END_IF

//To currents
	r_basecurrentSetpoint := LIMIT(-r_DynamicCurrentLimit, kWToCurrent(r_ActivePowerRQ, r_VoltAC), r_DynamicCurrentLimit);
	r_reactiveCurrentSetpoint := LIMIT(-fb_DynamicreactiveRemainMA.Q, kWToCurrent(r_ReactivePowerRQ,get.r_ACVoltageD7), fb_DynamicreactiveRemainMA.Q);	

//TO REFS
	r_InputActiveCurrentLimitRef := BaseValueToRef(r_InputActiveCurrentLimit);
	r_OutputActiveCurrentLimitRef := BaseValueToRef(r_OutputActiveCurrentLimit);
	r_baseCurrentRef := BaseValueToRef(r_basecurrentSetpoint);
	r_ReactivecurrentRef:= BaseValueToRef(r_reactiveCurrentSetpoint);

get.b_LimiterActive := TRUE;
// set limter state
IF r_ThrottlingValueMindex < fb_PIDMindex.fManSyncValue THEN
	get.e_ThrottlingStatus := ePowerModuleThrottlingState.Overvoltage;
ELSIF r_ThrottlingValueFilterTemp < r_MaxOvercurrentFactor THEN
	get.e_ThrottlingStatus := ePowerModuleThrottlingState.FilterTemp;
ELSIF r_ThrottlingValueInverterTemp < r_MaxOvercurrentFactor THEN
	get.e_ThrottlingStatus := ePowerModuleThrottlingState.InverterTemp;
ELSE
	get.b_LimiterActive := FALSE;
END_IF


	
//set the final value as feedback to the get struct of the powermodule
	get.r_OverCurrentValue 	:=  r_ThrottlingActual;
	get.r_Pmin 				:= -CurrentToKw(MIN(get.r_ACcurrentLimit, r_InputActiveCurrentLimit), r_VoltAC) * r_PLimitOverhead;
	get.r_Pmax 				:= CurrentToKw(MIN(get.r_ACcurrentLimit, r_outputActiveCurrentLimit), r_VoltAC);
	get.r_ACcurrentLimit	:= MIN(set.r_ACcurrentLimit, r_DynamicCurrentLimit);
	r_reactiveMaxCurrent 	:= MIN(fb_DynamicreactiveRemainMA.Q, SQRT(MAX(EXPT(get.r_ACcurrentLimit,2) - EXPT(get.r_ActiveCurrent,2), 0)));
	get.r_Qmax				:=  CurrentToKW(r_reactiveMaxCurrent, r_VoltAC);
	get.r_Qmin				:= -get.r_Qmax;
END_METHOD

METHOD PRIVATE SetInverterSettings : BOOL

VAR_INST
	ton_GridcodeOnDelay	: TON := (PT:= T#500MS);
	ton_GridcodeOffDelay: TON := (PT:= T#0S);
	SR_GridCodeActivate	: SR; 
	
	FtrigResetDrive		: F_TRIG;
END_VAR
//set actual droop
inverter.r_BaseRefRampRate		:= set.i_PowerChangeRate;

ton_GridcodeOffDelay(IN := (get.e_InverterMode <> eInvertermodes.Afe AND NOT get.GridcodeStatusWord.b_GridCodeTripActive) OR NOT get.StatusWord.b_Running);
ton_GridcodeOnDelay(IN:= get.e_InverterMode = eInvertermodes.Afe AND set.b_gridcodeEnable AND get.StatusWord.b_ReadyToOperate);
//Set gridcodes
SR_GridCodeActivate(
	SET1 := ton_GridcodeOnDelay.Q,
	RESET := ton_GridcodeOffDelay.Q OR NOT set.b_gridcodeEnable OR NOT get.StatusWord.b_ReadyToOperate,
	);


inverter.ControlWord.b_GridCodeEnable:= SR_GridCodeActivate.Q1;
inverter.controlword.b_ExtGridcodeTrip := set.b_ExtgridCodeTrip;

//reset drive if gridcodes are set off
FtrigResetDrive(CLK:= inverter.ControlWord.b_GridCodeEnable);
IF FtrigResetDrive.Q THEN
	Reset();
END_IF

IF NOT get.StatusWord.b_Running THEN
	//Set powermode
	inverter.Island(TRUE);
	//Set voltage / frequency
	//SetVoltageFrequency(TRUE, settings.GridParams.r_GridNominalVoltage, settings.GridParams.r_GridNominalFrequency);	
END_IF
END_METHOD

METHOD PRIVATE SetParallelDrive : BOOL
IF Settings.Configuration.b_DoublePowerModule THEN
	inverter.ControlWord.b_ParallelAFE := TRUE;
ELSE
	inverter.ControlWord.b_ParallelAFE:= FALSE;
END_IF

SetParallelDrive := Settings.Configuration.b_DoublePowerModule;
END_METHOD

METHOD SetVoltageFrequency : BOOL
VAR_INPUT
	SetToIn		: BOOL;
	VoltIN		: REAL;
	FreqIN		: REAL;
END_VAR

VAR_INST
	//rTrig_SetToIN	: R_TRIG;
END_VAR

VAR_INST
	r_FrequencyDroopOffset 	: REAL;
	r_VoltageDroopOffset 	: REAL;
	//freqRamp				: FB_ramp := (b_enable := TRUE, r_rampRate := 10);
	//VoltRamp				: FB_ramp := (b_enable := TRUE, r_rampRate := 10);
END_VAR
//rTrig_SetToIN(CLK := SetToIn);
//FreqRamp(SetToIn := NOT get.StatusWord.b_Running OR rTrig_SetToIN.Q);
//VoltRamp(SetToIn := NOT get.StatusWord.b_Running OR rTrig_SetToIN.Q);
//FreqRamp.IN := FreqIN;	
//VoltRamp.IN := VoltIN;

// set gridnominal Frequency
r_FrequencyDroopOffset := FreqIN - settings.GridParams.r_GridNominalFrequency;
inverter.r_FrequencyDroopOffset := LIMIT(-2, r_FrequencyDroopOffset, 2);
// set gridnominal voltage
r_VoltageDroopOffset := VoltIN - settings.GridParams.r_GridNominalVoltage + st_params.i_VoltageOffset;
inverter.r_VoltageCorrection	:= LIMIT(-40 + st_params.i_VoltageOffset, r_VoltageDroopOffset, 40 + st_params.i_VoltageOffset);
END_METHOD

METHOD Shutdown : BOOL
VAR_INPUT
	b_Force		: BOOL := FALSE;
END_VAR

VAR_INST
	b_enableForce : BOOL := FALSE;
	currentMax : REAL;
	r_DCcurrentAbs : REAL;
	r_DCcurrent	: REAL;
END_VAR

VAR
	r_DCreleaseCurrent		: REAL := 20;
END_VAR
r_DCcurrentAbs := ABS(get.r_DCCurrent);
inverter.r_BaseCurrentRef := 0;
inverter.r_ReactiveCurrentRef := 0;

IF (b_Force OR get.StatusWord.b_Fault) THEN
	inverter.ControlWord.b_ChargeDC := FALSE;
	inverter.ControlWord.b_run := FALSE;
ELSE
	inverter.ControlWord.b_run := FALSE;
	inverter.r_OutputActiveCurrentLimit := 10;
	inverter.r_InputActiveCurrentLimit := 10;
	IF r_DCcurrentAbs < r_DCreleaseCurrent THEN
		inverter.ControlWord.b_ChargeDC := FALSE;
		buscoupler.b_MCCBChargeSpring := TRUE;	
	END_IF
END_IF

//minimum shutdown execution time.
shutdown := NOT inverter.ControlWord.b_ChargeDC AND NOT inverter.ControlWord.b_run AND NOT get.StatusWord.b_Running AND DecoupleDC();
END_METHOD

METHOD Start : BOOL

VAR_INPUT
	AFESTART : BOOL;
END_VAR

VAR_INST
	tp_RunDelay			: TP := (PT:= T#1S);
	StartupValue		:	BOOL := TRUE;
	b_RunAlready		: BOOl;
END_VAR
inverter.r_OutputActiveCurrentLimit := 520;
inverter.r_InputActiveCurrentLimit := 520; 
inverter.ControlWord.b_run := FALSE;
inverter.startMode := TRUE;

IF AFESTART THEN
	inverter.AFE();
ELSE
	inverter.Island(TRUE);
END_IF

SetVoltageFrequency(TRUE, settings.GridParams.r_GridNominalVoltage, settings.GridParams.r_GridNominalFrequency);

(*STEPS
first check if DC exists
if its yet there and checkDCvoltage gives TRUE, inverter can get to run state.
Ifnot, try precharging (if its in the system).

*)
IF get.b_MccbUvr24VdcOK THEN
	inverter.ControlWord.b_ChargeDC := get.StatusWord.b_ReadyToDCCharge;
	tp_RunDelay(in := CheckDCvoltage() AND NOT tp_RunDelay.Q);
	b_RunAlready := get.StatusWord.b_running AND get.r_ACVoltageSupply <> 0;
	inverter.ControlWord.b_run := tp_RunDelay.Q OR b_RunAlready;
END_IF


//Check if we already have DC
IF CoupleDC() THEN
	Start := get.StatusWord.b_Running;
END_IF



//OLD code, run delay and startup value might be needed -- To be tested
(*


IF CheckDCvoltage(r_BatDcVoltage) THEN
	inverter.ControlWord.b_ChargeDC := get.StatusWord.b_ReadyToDCCharge;
	inverter.ControlWord.b_run := tp_RunDelay.Q OR startupValue;
	StartupValue := FALSE;
	
	IF get.StatusWord.b_Running THEN
		tp_RunDelay(in := FALSE);
	END_IF
	Start := get.StatusWord.b_Running;
END_IF
*)
END_METHOD

END_FUNCTION_BLOCK

(* stored: Version 1.1.0.1, ProductVersion 3.1.4024.12
   POU FB_PowerModule: Id {a42b7ccb-ca12-4e75-939b-ec7736ea81fa}, SpecialFunc None
   Folder Private: Id {4be62864-28d1-4476-8537-b9c9cd92a6c0}
   Method BaseValueToRef: Id {2b120fb5-7ad4-425b-835d-ff7a0fcb459b}
   Method CalculateDerivativePowerValues: Id {e9b79040-160b-44bf-b42e-34ec5550e0ac}
   Method CheckDCVoltage: Id {83d8481d-d542-4722-93fb-a950ab9b03d2}
   Method CompensationCurve: Id {bc751060-4b54-4af7-bec9-61ddf2be36d2}
   Method CoupleDC: Id {f6b1267e-4b37-4141-b5dd-1f04ceab32d7}
   Method DecoupleDC: Id {80672981-1c50-4852-b65c-7652fd61c115}
   Method FanControl: Id {d7f433ac-9a45-40cb-a569-72ac94992e76}
   Method FillAdditionalGets: Id {1853e9dc-cf20-4497-9be4-cf8b77465570}
   Method GetDiagnostics: Id {2f1d3e3d-eacf-4f40-bc7d-70dee9f4b860}
   Method GetInverterModes: Id {d81a850a-25c1-4f3c-9483-87bd52313c5b}
   Method GetMaxTemperature: Id {a1e4f906-4640-420c-84ca-155f010e48e2}
   Method GetPowerModuleStatus: Id {d7999da7-9ef9-4a4c-98e2-5186b30148b6}
   Method GetTemperatureEvents: Id {35c96a1b-0afe-4178-a1de-7b941b5c2c12}
   Method Idle: Id {8d015fbe-2d0a-4a27-abbf-72693d9cf6a0}
   Method init: Id {cf76f424-9635-468b-b6d4-81f8cfce1a5c}
   Method Reset: Id {110855c6-4caf-42ad-88b8-66286c4b2542}
   Method Run: Id {cbd44e23-f9bb-4d57-8fcc-99d8fc41d5c4}
   Method SetEvents: Id {d0c0a999-9eca-43ec-856e-48bb80c84e53}
   Method SetInverterRefs_Limits: Id {f3ee8422-a69b-4266-b405-ac58a0ba67e6}
   Method SetInverterSettings: Id {6b2cda43-5f42-41e4-9aff-67f9295db7ea}
   Method SetParallelDrive: Id {515f6b75-056f-440d-be15-5fab4dd82664}
   Method SetVoltageFrequency: Id {d2ca8923-fabe-415e-bbcb-3e5e102161ea}
   Method Shutdown: Id {16e88d59-8ee2-4197-a519-fb96d1af3315}
   Method Start: Id {85e42802-1b0b-4902-9b56-8a9abd9dcaba} *)
